INTERFACE I_VisitIntances

METHOD PUBLIC Visit
VAR_INPUT
	Instance : I_Instance;
END_VAR
END_METHOD

END_INTERFACE

(* stored: Version 1.1.0.1, ProductVersion 3.1.4024.11
   Itf I_VisitIntances: Id {2024b737-6a84-48f4-baeb-093a18ac9cb0}
   Method Visit: Id {08f06157-7fef-4f58-9f10-d92841ef6b0a} *)
